PROGRAM PRG_Test
VAR
	validateFunctionsTest : ValidateFunctionsTest;
	manipulateFunctionsTest : ManipulateFunctionsTest;
	convertFunctionsTest : ConvertFunctionsTest;
	
	sb255Test : StringBuilder255Test;
	buildStringInlineTest : BuildStringInlineTest;
	sbExtBufferTest : StringBuilderExtBufferTest;
	sbInfiniteTest : StringBuilderInfiniteTest;
END_VAR

TcUnit.RUN();

END_PROGRAM

(* stored: Version 1.1.0.1, ProductVersion 3.1.4024.12
   POU PRG_Test: Id {93887d91-9466-4bc5-b21d-06b0d85b60ea}, SpecialFunc None *)
